TYPE CAR :
STRUCT
	pX : REAL;
	pY : REAL;
	currentTrack : SINT:=1;
	//queueNum : DINT;
	carID : SINT;
	present: BOOL;
	percentFull: REAL;
	positionID: INT;
	fwdCMD: BOOL;
	revCMD: BOOL;
	initCar: BOOL;
	isAttached: BOOL;
	isOnBOardRed: BOOL;
	isOnBoardBlue: BOOL;
	cmdAttach: BOOL;
	cmdDetach: BOOL;
	
END_STRUCT
END_TYPE

(* stored: Version 1.1.0.1
   DUT CAR: Id {903b4816-ae89-40d5-8573-3632da433666} *)
